Universal Robots PolyScope program: head_turn_on.urp

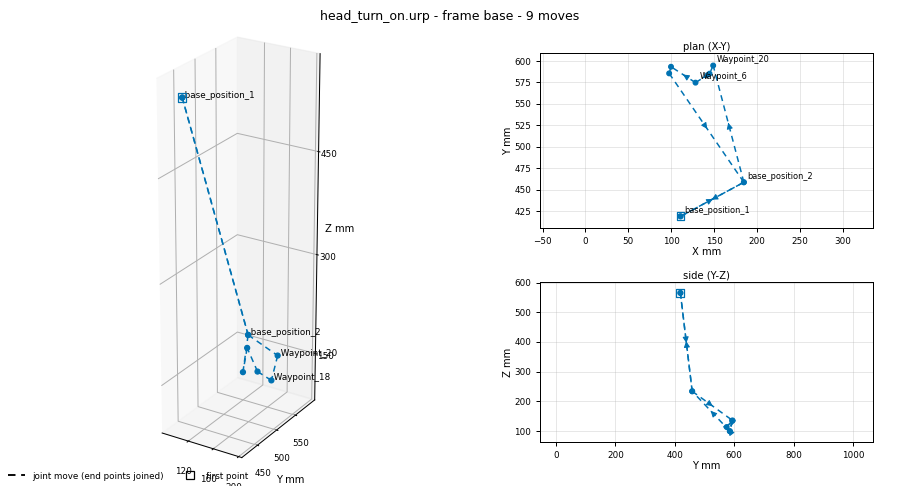
[picture p0: tool path of head_turn_on.urp in frame base, 9 of 9 moves have a stored position in this frame; points joined in program order, loops and branches not executed]
Program head_turn_on (installation=default directory=/programs/Nicolas_Arteaga/quality createdIn=5.12.4.1101661 lastSavedIn=5.12.4.1101661 robotSerialNumber=20225502378)
Calibrated DH parameters: a=[0.00022, -0.425328, -0.389701, 0.000059, 0.000065, 0]; d=[0.162608, 0.803456, 9.992211, -10.662202, 0.099702, 0.099559]; alpha=[1.570756, 0.001543, 0.004316, 1.570651, -1.570122, 0]; deltaTheta=[0, 0.002917, 0.116094, -0.119008, 0, -0.000001]
Robot Program (runOnlyOnce=true)
  'Turns on the heat and the motor'
  MoveJ speed 60 deg/s, acceleration 80 deg/s^2 (useActiveTCP=true) feature=Base
    Waypoint base_position_1: TCP in base x=110.873 y=418.875 z=565.206 mm, rx=-1.5602 ry=-0.9891 rz=-1.3624 rad; joints [200.91, -129.117, 99.415, 36.172, 41.428, 90] deg; TCP offset x=0 y=0 z=191.5 mm, rx=0 ry=0 rz=0 rad
    URCap Gripper Activate (Robotiq_Grippers, Robotiq Inc.) dataModel(ResetAndActivateKey=false)
    URCap Gripper (Robotiq_Grippers, Robotiq Inc.) dataModel(position=100.0, force=0.0, speed=100.0, positionInDouble=100.0, forceInDouble=0.0, speedInDouble=100.0, slaveIds=[9], blocking=true)
    Waypoint base_position_2: TCP in base x=184.715 y=458.614 z=234.006 mm, rx=-1.6866 ry=-0.757 rz=-1.7388 rad; joints [237.954, -104.402, 143.977, -41.546, 99.477, 90] deg; TCP offset x=0 y=0 z=191.5 mm, rx=0 ry=0 rz=0 rad
    Waypoint Waypoint_20: TCP in base x=148.965 y=594.736 z=135.542 mm, rx=-1.534 ry=-0.9908 rz=-1.4978 rad; joints [241.135, -76.483, 134.799, -57.047, 85.473, 90.096] deg; TCP offset x=0 y=0 z=191.5 mm, rx=0 ry=0 rz=0 rad
    Waypoint Waypoint_18: TCP in base x=144.729 y=585.254 z=99.641 mm, rx=-1.6452 ry=-1.0629 rz=-1.3952 rad; joints [240.345, -76.212, 134.041, -48.93, 84.034, 89.956] deg
    Waypoint Waypoint_6: TCP in base x=128.361 y=574.771 z=113.603 mm, rx=-1.6021 ry=-1.0547 rz=-1.4085 rad; joints [240.991, -78.96, 136.832, -51.045, 83.741, 89.995] deg
    Waypoint Waypoint_17: TCP in base x=99.779 y=593.316 z=135.031 mm, rx=-1.492 ry=-1.1083 rz=-1.3373 rad; joints [241.005, -80.644, 135.434, -49.386, 76.736, 90.11] deg
    Waypoint Waypoint_16: TCP in base x=97.63 y=585.581 z=99.564 mm, rx=-1.5888 ry=-1.15 rz=-1.2562 rad; joints [240.815, -78.841, 134.769, -44.332, 76.722, 90.097] deg
    Waypoint base_position_2: TCP in base x=184.715 y=458.614 z=234.006 mm, rx=-1.6866 ry=-0.757 rz=-1.7388 rad; joints [237.954, -104.402, 143.977, -41.546, 99.477, 90] deg; TCP offset x=0 y=0 z=191.5 mm, rx=0 ry=0 rz=0 rad
    Waypoint base_position_1: TCP in base x=110.873 y=418.875 z=565.206 mm, rx=-1.5602 ry=-0.9891 rz=-1.3624 rad; joints [200.91, -129.117, 99.415, 36.172, 41.428, 90] deg; TCP offset x=0 y=0 z=191.5 mm, rx=0 ry=0 rz=0 rad
